// TIA Portal V19 export
DATA_BLOCK "DI_FW_MANAGER"   // DB10
AUTHOR : MS
// stored: AutoNumber false, InstanceOfName FB_FW_MANAGER, InstanceOfType FB
"FB_FW_MANAGER"
   // VAR_INPUT
   //    CallDBNr : DB_ANY := 22;
   // END_VAR
   // VAR RETAIN
   //    leng : Int := 18;
   //    Offset : Int := 50;
   //    resDW_1 : DWord := 16#0000_0000;
   //    resDW_2 : DWord := 16#0000_0000;
   //    resDW_3 : DWord := 16#0000_0000;
   //    resDW_4 : DWord := 16#0000_0000;
   //    Kettenpos : Array[1..4] of Byte;
   //    Auto : Struct
   //       Anlage : Bool := FALSE;
   //       Reihe_1 : Bool := FALSE;
   //       Reihe_2 : Bool := FALSE;
   //       Reihe_3 : Bool := FALSE;
   //       Reihe_4 : Bool := FALSE;
   //       Reihe_5 : Bool := FALSE;
   //       res : Bool := FALSE;
   //       res_1 : Bool := FALSE;
   //       Anlage_not : Bool := TRUE;
   //       Reihe_not_1 : Bool := TRUE;
   //       Reihe_not_2 : Bool := FALSE;
   //       Reihe_not_3 : Bool := FALSE;
   //       Reihe_not_4 : Bool := FALSE;
   //       Reihe_not_5 : Bool := FALSE;
   //       res_2 : Bool := FALSE;
   //       res_3 : Bool := FALSE;
   //    END_STRUCT;
   //    resDW_6 : DWord := 16#0000_0000;
   //    resDW_7 : DWord := 16#0000_0000;
   //    resDW_8 : DWord := 16#0000_0000;
   //    resDW_9 : DWord := 16#0000_0000;
   //    resW : Int := 0;
   //    akt_CT : Int := 26;
   //    max_CT : Int := 41;
   //    FW_DAT : Array[1..20] of Struct
   //       WT_NR_LANG : DInt;
   //       IST_POS : Byte;
   //       ZIEL_POS : Byte;
   //       Fahrt_Vor : Bool;
   //       Fahrt_Rck : Bool;
   //       Heben : Bool;
   //       Senken : Bool;
   //       Bereit : Bool;
   //       Fehler : Bool;
   //       Dummy : Bool;
   //       res : Bool;
   //       Tipp : Bool;
   //       Hand : Bool;
   //       Auto_Stop : Bool;
   //       Auto : Bool;
   //       Halt : Bool;
   //       K_Auto : Bool;
   //       Kette_wait_Start : Bool;
   //       Kette_wait_Ende : Bool;
   //       Unten : Bool;
   //       Z_Sensor : Bool;
   //       Oben : Bool;
   //       mittig : Bool;
   //       HWmittig : Bool;
   //       res_7 : Bool;
   //       res_8 : Bool;
   //       res_9 : Bool;
   //       WT_DB_Nr : Byte;
   //       IstInc : DInt;
   //       Stangen_Nr : Byte;
   //       WT_Typ : Byte;
   //       priorisirt : Bool;
   //       in_Anlage : Bool;
   //       in_Entmetall : Bool;
   //       aus_Anlage : Bool;
   //       aus_Entmetall : Bool;
   //       Speicherprog : Bool;
   //       Trommel : Bool;
   //       Leer_WT : Bool;
   //       BefX : Byte;
   //    END_STRUCT;
   // END_VAR
BEGIN
   Kettenpos[1..4] := 16#00;
   FW_DAT[1..20].WT_NR_LANG := 0;
   FW_DAT[1].IST_POS := 16#02;
   FW_DAT[2].IST_POS := 16#0B;
   FW_DAT[3].IST_POS := 16#2C;
   FW_DAT[4].IST_POS := 16#4A;
   FW_DAT[5].IST_POS := 16#02;
   FW_DAT[6].IST_POS := 16#2F;
   FW_DAT[7..20].IST_POS := 16#00;
   FW_DAT[1..20].ZIEL_POS := 16#00;
   FW_DAT[1..20].Fahrt_Vor := FALSE;
   FW_DAT[1..20].Fahrt_Rck := FALSE;
   FW_DAT[1..20].Heben := FALSE;
   FW_DAT[1..20].Senken := FALSE;
   FW_DAT[1..6].Bereit := TRUE;
   FW_DAT[7..20].Bereit := FALSE;
   FW_DAT[1..20].Fehler := FALSE;
   FW_DAT[1..20].Dummy := FALSE;
   FW_DAT[1..20].res := FALSE;
   FW_DAT[1..20].Tipp := FALSE;
   FW_DAT[1..6].Hand := TRUE;
   FW_DAT[7..20].Hand := FALSE;
   FW_DAT[1..20].Auto_Stop := FALSE;
   FW_DAT[1..20].Auto := FALSE;
   FW_DAT[1..20].Halt := FALSE;
   FW_DAT[1..6].K_Auto := TRUE;
   FW_DAT[7..20].K_Auto := FALSE;
   FW_DAT[1..4].Kette_wait_Start := TRUE;
   FW_DAT[5..20].Kette_wait_Start := FALSE;
   FW_DAT[1..4].Kette_wait_Ende := TRUE;
   FW_DAT[5..20].Kette_wait_Ende := FALSE;
   FW_DAT[1..4].Unten := TRUE;
   FW_DAT[5..20].Unten := FALSE;
   FW_DAT[1..20].Z_Sensor := FALSE;
   FW_DAT[1..20].Oben := FALSE;
   FW_DAT[1..6].mittig := TRUE;
   FW_DAT[7..20].mittig := FALSE;
   FW_DAT[1..20].HWmittig := FALSE;
   FW_DAT[1..20].res_7 := FALSE;
   FW_DAT[1..20].res_8 := FALSE;
   FW_DAT[1..20].res_9 := FALSE;
   FW_DAT[1..20].WT_DB_Nr := 16#00;
   FW_DAT[1].IstInc := 1998;
   FW_DAT[2].IstInc := 10998;
   FW_DAT[3].IstInc := 43999;
   FW_DAT[4].IstInc := 49759;
   FW_DAT[5..20].IstInc := 0;
   FW_DAT[1..20].Stangen_Nr := 16#00;
   FW_DAT[1..20].WT_Typ := 16#00;
   FW_DAT[1..20].priorisirt := FALSE;
   FW_DAT[1..20].in_Anlage := FALSE;
   FW_DAT[1..20].in_Entmetall := FALSE;
   FW_DAT[1..20].aus_Anlage := FALSE;
   FW_DAT[1..20].aus_Entmetall := FALSE;
   FW_DAT[1..20].Speicherprog := FALSE;
   FW_DAT[1..20].Trommel := FALSE;
   FW_DAT[1..20].Leer_WT := FALSE;
   FW_DAT[1..20].BefX := 16#00;
END_DATA_BLOCK
